Fanuc KAREL source: kb00088.KL

-- PROVISIONAL review KL for V1013-1; original PC SHA256 4d621db8a54fb15987ea48bee3d3dd521ecd30352c9de5e43ff51603b7553613
-- Incomplete behavior may be omitted. Consult companion uncertainty JSON. Do not deploy.
PROGRAM KB00088
%NOLOCKGROUP
BEGIN
  -- UNRESOLVED_PC offsets 5-12; opcodes 9D,23
  -- UNRESOLVED_PC offsets 17-24; opcodes 9D,23
  -- UNRESOLVED_PC offsets 29-36; opcodes 9D,23
  -- UNRESOLVED_PC offsets 41-77; opcodes 27,22,22,22,27,9D,31,7E,4A
  -- UNRESOLVED_PC offsets 82-86; opcodes 7F
END KB00088
